//==================================================================================================
//								RJM Maszyny sp. z o.o.
//									13.05.2022
//	Obsluga przesuwacza na siłowniku 
//	Siłownik zabieraka plus siłownik przesuwający 
//	Cykl przesuwania: wysun zabierak -> przesun -> schowaj zabierak -> powrót  
// 	v1.0	|| TC v 3.1.4024.22		|| - pierwsza wersja
//==================================================================================================
FUNCTION_BLOCK FB_PrzesuwaczNaSilowniku
VAR_INPUT
	stParametry								: DUT_PrzesuwaczNaSilowniku_Parametry;
END_VAR
VAR_OUTPUT
END_VAR
VAR
	bCzujnik0Zabieraka						: ITF_Czujnik;
	bCzujnikMaxZabieraka					: ITF_Czujnik;
	fbElektrozaworZabieraka					: ITF_Elektozawor;
	bCzujnik0Przesuwacza					: ITF_Czujnik;
	bCzujnikMaxPrzesuwacza					: ITF_Czujnik;
	fbElektrozaworPrzesuwacza				: ITF_Elektozawor;
	fbZabierak								: FB_Silownik_Kontola (fbCzujnikPozycja0 		:= bCzujnik0Zabieraka, 
																	fbCzujnikPozycjaMax 	:= bCzujnikMaxZabieraka,
																	fbElektrozawor 			:= fbElektrozaworZabieraka);
	fbPrzesuwaczNaped						: FB_Silownik_Kontola (fbCzujnikPozycja0 		:= bCzujnik0Przesuwacza, 
																	fbCzujnikPozycjaMax 	:= bCzujnikMaxPrzesuwacza,
																	fbElektrozawor 			:= fbElektrozaworPrzesuwacza);	
	arrElementyWykonawcze 					: ARRAY [1..10] OF ITF_LogowanieBledow_ElementWykonawczy := 
														[fbZabierak.fbLBKomunikacja, 
														fbPrzesuwaczNaped.fbLBKomunikacja];
	fbLBKomunikacja							: FB_PrzesuwaczNaSilowniku_Komunikacja 
														(arrElementyWykonawcze := arrElementyWykonawcze,
														iIloscPodlementow := 2);
	bWykonajCyklPrzesuwania					: BOOL;
	bCyklPrzesuwania						: BOOL;
	bCyklPrzesuWaniaSkonczony				: BOOL;
	bBazuj									: BOOL;
	bBazowanie								: BOOL;
	bCyklBazowaniaSkonczony					: BOOL;
	bReset									: BOOL;
	bPierwszePrzejscieBazowanie				: BOOL;
	bPierwszePrzejsciePrzesuwanie			: BOOL;
	iKrokPrzesuwania						: INT := 0;
	tonChwilaPoDojechaniu					: TON;
END_VAR

PROPERTY Bazowanie : BOOL
GET
Bazowanie									:= bBazuj;
END_GET
END_PROPERTY

PROPERTY Bazuj : BOOL
SET
bBazuj										:= Bazuj;
END_SET
END_PROPERTY

METHOD PRIVATE CyklBazowania_Praca : BOOL
VAR_INPUT
END_VAR
IF (NOT bPierwszePrzejscieBazowanie) THEN
	bPierwszePrzejscieBazowanie				:= TRUE;
	bCyklBazowaniaSkonczony					:= FALSE;
	fbZabierak.PrzesunDoPoczatku			:= TRUE;
END_IF

IF (fbZabierak.NaPoczatku AND NOT fbPrzesuwaczNaped.PrzesuwanieWStronePoczatku) THEN
	fbPrzesuwaczNaped.PrzesunDoPoczatku		:= TRUE;
END_IF

IF (fbPrzesuwaczNaped.NaPoczatku AND fbZabierak.NaPoczatku) THEN
	bPierwszePrzejscieBazowanie				:= FALSE;
	bCyklBazowaniaSkonczony					:= TRUE;
	CyklBazowania_Praca						:= TRUE;
ELSE
	CyklBazowania_Praca						:= FALSE;
END_IF
END_METHOD

PROPERTY CyklPrzesuwania : BOOL
GET
CyklPrzesuwania								:= bCyklPrzesuwania;
END_GET
END_PROPERTY

METHOD CyklPrzesuwania_Praca : BOOL
VAR_INPUT
END_VAR
IF (NOT bPierwszePrzejsciePrzesuwanie) THEN
	bPierwszePrzejsciePrzesuwanie			:= TRUE;
	bCyklPrzesuWaniaSkonczony				:= FALSE;
	fbZabierak.PrzesunDoKonca				:= TRUE;
	tonChwilaPoDojechaniu.IN				:= FALSE;
	iKrokPrzesuwania						:= 1;
END_IF

CASE iKrokPrzesuwania OF
	1	:
	IF (fbZabierak.NaKoncu) THEN
		fbPrzesuwaczNaped.PrzesunDoKonca	:= TRUE;
		iKrokPrzesuwania					:= 10;
		CyklPrzesuwania_Praca				:= TRUE;
	END_IF
	10	:
	IF (fbPrzesuwaczNaped.NaKoncu) THEN
		tonChwilaPoDojechaniu.IN			:= TRUE;
		iKrokPrzesuwania					:= 20;
		CyklPrzesuwania_Praca				:= TRUE;
	END_IF
	20	:
	IF (tonChwilaPoDojechaniu.Q) THEN
		tonChwilaPoDojechaniu.IN			:= FALSE;
		fbZabierak.PrzesunDoKonca			:= TRUE;
		iKrokPrzesuwania					:= 30;
		CyklPrzesuwania_Praca				:= TRUE;
	END_IF
	30	:
	IF (fbZabierak.NaPoczatku) THEN
		fbPrzesuwaczNaped.PrzesunDoPoczatku	:= TRUE;
		iKrokPrzesuwania					:= 40;
		CyklPrzesuwania_Praca				:= TRUE;
	END_IF
	40	:
	IF (fbPrzesuwaczNaped.NaPoczatku) THEN
		iKrokPrzesuwania					:= 50;
		CyklPrzesuwania_Praca				:= TRUE;
		bCyklPrzesuWaniaSkonczony			:= TRUE;
	END_IF
	50	:
		iKrokPrzesuwania					:= 0;
		CyklPrzesuwania_Praca				:= FALSE;
END_CASE
END_METHOD

PROPERTY CyklPrzesuWaniaSkonczony : BOOL
GET
CyklPrzesuWaniaSkonczony					:= bCyklPrzesuWaniaSkonczony;
END_GET
END_PROPERTY

METHOD FB_init : BOOL
VAR_INPUT
	bInitRetains : BOOL; // if TRUE, the retain variables are initialized (warm start / cold start)
	bInCopyCode : BOOL;  // if TRUE, the instance afterwards gets moved into the copy code (online change)
	bCzujnik0Zabieraka						: ITF_Czujnik;
	bCzujnikMaxZabieraka					: ITF_Czujnik;
	fbElektrozaworZabieraka					: ITF_Elektozawor;
	bCzujnik0Przesuwacza					: ITF_Czujnik;
	bCzujnikMaxPrzesuwacza					: ITF_Czujnik;
	fbElektrozaworPrzesuwacza				: ITF_Elektozawor;
END_VAR
THIS^.bCzujnik0Zabieraka					:= bCzujnik0Zabieraka;			     
THIS^.bCzujnikMaxZabieraka					:= bCzujnikMaxZabieraka;		    
THIS^.fbElektrozaworZabieraka				:= fbElektrozaworZabieraka;		 
THIS^.bCzujnik0Przesuwacza					:= bCzujnik0Przesuwacza;		    
THIS^.bCzujnikMaxPrzesuwacza				:= bCzujnikMaxPrzesuwacza;		  
THIS^.fbElektrozaworPrzesuwacza				:= fbElektrozaworPrzesuwacza;

THIS^.fbZabierak.FB_init (FALSE, FALSE, bCzujnik0Zabieraka, bCzujnikMaxZabieraka, fbElektrozaworZabieraka);
THIS^.fbPrzesuwaczNaped.FB_init (FALSE, FALSE, bCzujnik0Przesuwacza, bCzujnikMaxPrzesuwacza, fbElektrozaworPrzesuwacza);
END_METHOD

METHOD Praca : BOOL
VAR_INPUT
END_VAR
//---------------Resetowanie zmiennych
	IF (bReset) THEN
		Resetowanie ();
	END_IF
//---------------Resetowanie zmiennych
//---------------Bazowanie siłowników - powrót do poczatku
	IF (bBazuj) THEN
		bBazowanie								:= TRUE;
	END_IF
	IF (bBazowanie) THEN
		bBazowanie								:= CyklBazowania_Praca ();
	END_IF
//---------------Bazowanie siłowników - powrót do poczatku
//---------------Cykl przesuwnaia - koniec gora dol poczatek
	IF (bWykonajCyklPrzesuwania) THEN
		bCyklPrzesuwania						:= TRUE;
	END_IF
	tonChwilaPoDojechaniu (PT := REAL_TO_TIME (stParametry.rCzasNaKoncu));
	IF (bCyklPrzesuwania) THEN
		bCyklPrzesuwania						:= CyklPrzesuwania_Praca ();
	END_IF
//---------------Cykl przesuwnaia - koniec gora dol poczatek
END_METHOD

METHOD PRIVATE Resetowanie : BOOL
VAR_INPUT
END_VAR
bWykonajCyklPrzesuwania						:= FALSE;
bCyklPrzesuwania							:= false;
bCyklPrzesuWaniaSkonczony					:= false;
bBazuj										:= false;
bBazowanie									:= false;
bCyklBazowaniaSkonczony						:= FALSE;
bPierwszePrzejscieBazowanie					:= FALSE;
bPierwszePrzejsciePrzesuwanie				:= FALSE;
tonChwilaPoDojechaniu.IN					:= FALSE;


bReset										:= FALSE;
END_METHOD

PROPERTY Resetuj : BOOL
SET
bReset										:=Resetuj;
END_SET
END_PROPERTY

PROPERTY WykonajCyklPrzesuwania : BOOL
SET
bWykonajCyklPrzesuwania						:= WykonajCyklPrzesuwania;
END_SET
END_PROPERTY

END_FUNCTION_BLOCK

(* stored: Version 1.1.0.1, ProductVersion 3.1.4024.11
   POU FB_PrzesuwaczNaSilowniku: Id {c7ba1278-3548-4e13-8976-321b6c21dbe0}, SpecialFunc None
   Property Bazowanie: Id {ea84dae0-db67-4001-9f56-c7d50c87da36}
   Get Get: Id {8990b3c0-edfa-4aa4-aa06-b75bbd90f054}
   Property Bazuj: Id {48299f66-cf2b-4f41-bd89-ab4fd693cdf8}
   Set Set: Id {c2df6c92-4390-4584-947f-0489e3c91278}
   Method CyklBazowania_Praca: Id {e436b484-17c0-47ed-a727-72ecc434ecc6}
   Property CyklPrzesuwania: Id {9dbd02be-7b8b-4bc5-881c-396938a1e639}
   Get Get: Id {362a1c75-df31-419f-9ede-ed576cdc01f3}
   Method CyklPrzesuwania_Praca: Id {c5710e17-cb66-4931-8ad1-c66f04ccc386}
   Property CyklPrzesuWaniaSkonczony: Id {67556867-1f57-4eb1-a7b8-fe1b44636d00}
   Get Get: Id {c849afb2-5ecd-4244-9b25-a1e4a3a4edda}
   Method FB_init: Id {1ce11768-98bf-4742-be1e-5a2040e34f8c}
   Method Praca: Id {44cee759-01b2-476e-b3ae-9fcfed73cbf4}
   Method Resetowanie: Id {3266a3b4-85c7-4870-b306-21ac7a9cbdf6}
   Property Resetuj: Id {da194d34-255f-4986-bd5f-ef9469dd78f1}
   Set Set: Id {01fa9a79-b8bf-4b07-b476-18d11ab8ba51}
   Property WykonajCyklPrzesuwania: Id {ae9011c0-d4ee-453e-b80c-6b486d3263af}
   Set Set: Id {4d65ef21-a11d-49b0-9652-ef6880dd4a1b} *)
